(* CODESYS project EL6224_Youtube_Lib.library
   Title: myLibrary
   Version: 0.2
   Placeholder: myLibrary
   Company: soup01

Project tree, tasks and I/O mapping:
  libraries: Tc2_Standard, * (Beckhoff Automation GmbH); Tc2_System, * (Beckhoff Automation GmbH); Tc3_IoLink, * (Beckhoff Automation GmbH); Tc3_Module, * (Beckhoff Automation GmbH); VisuSymbols, 3.5.10.0 (System)
  DUTs/
    data type DUT_ATV320_HMI_NW3_4_PL
    interface ITF_EL6224_Basic: METH_Port_OK
    interface ITF_IDWE_M12MM_NMS_A0: METH_Disable, METH_Update, Prop_ALR, Prop_ALR1, Prop_ALR2, Prop_ALR3, Prop_Enable, Prop_MeasurementValue, Prop_OSS1, Prop_OSS2, Prop_ScalingValue, Prop_StatusWord, Prop_TSS
    interface ITF_LR_TB2000: METH_Update, Prop_Distance, Prop_Enable
  GVLs/
  POUs/
    function block FB_EL6224_Basic [ST]: METH_Port_OK
    function block FB_IDWE_M12MM_NMS_A0 [ST]: METH_Disable, METH_Update, Prop_ALR, Prop_ALR1, Prop_ALR2, Prop_ALR3, Prop_Enable, Prop_MeasurementValue, Prop_OSS1, Prop_OSS2, Prop_ScalingValue, Prop_StatusWord, Prop_TSS
    function block FB_LR_TB2000 [ST]: METH_Update, Prop_Distance, Prop_Enable
  VISUs/
  text list GlobalTextList
*)

// DUTs/DUT_ATV320_HMI_NW3_4_PL
TYPE DUT_ATV320_HMI_NW3_4_PL:
STRUCT
	DIs		:ARRAY[1..6]OF BOOL;
	STO		:BOOL;
END_STRUCT
END_TYPE

// DUTs/ITF_EL6224_Basic
INTERFACE ITF_EL6224_Basic

METHOD METH_Port_OK : BOOL
VAR_INPUT
	iPort		:INT;
END_VAR
END_METHOD

END_INTERFACE

// DUTs/ITF_IDWE_M12MM_NMS_A0
INTERFACE ITF_IDWE_M12MM_NMS_A0

METHOD METH_Disable : BOOL
VAR_INPUT
	iTrigger		:BOOL;
END_VAR
END_METHOD

METHOD METH_Update : BOOL
END_METHOD

PROPERTY Prop_ALR : BOOL
GET
END_GET
END_PROPERTY

PROPERTY Prop_ALR1 : BOOL
GET
END_GET
END_PROPERTY

PROPERTY Prop_ALR2 : BOOL
GET
END_GET
END_PROPERTY

PROPERTY Prop_ALR3 : BOOL
GET
END_GET
END_PROPERTY

PROPERTY Prop_Enable : BOOL
GET
END_GET
END_PROPERTY

PROPERTY Prop_MeasurementValue : INT
GET
END_GET
END_PROPERTY

PROPERTY Prop_OSS1 : BOOL
GET
END_GET
END_PROPERTY

PROPERTY Prop_OSS2 : BOOL
GET
END_GET
END_PROPERTY

PROPERTY Prop_ScalingValue : Byte
GET
END_GET
END_PROPERTY

PROPERTY Prop_StatusWord : byte
GET
END_GET
END_PROPERTY

PROPERTY Prop_TSS : BOOL
GET
END_GET
END_PROPERTY

END_INTERFACE

// DUTs/ITF_LR_TB2000
INTERFACE ITF_LR_TB2000

METHOD METH_Update : BOOL
VAR_INPUT
END_VAR
END_METHOD

PROPERTY Prop_Distance : INT
GET
END_GET
END_PROPERTY

PROPERTY Prop_Enable : BOOL
GET
END_GET
END_PROPERTY

END_INTERFACE

// POUs/FB_EL6224_Basic
FUNCTION_BLOCK FB_EL6224_Basic IMPLEMENTS ITF_EL6224_Basic
VAR_INPUT
END_VAR
VAR_OUTPUT
END_VAR
VAR
	DeviceStatesInputs	AT %I*:ARRAY[1..4]OF USINT;
END_VAR

METHOD METH_Port_OK : BOOL
VAR_INPUT
	iPort	: INT;
END_VAR

METH_Port_OK:=FALSE;

CASE iPort OF
	1..4:
		METH_Port_OK:=DeviceStatesInputs[iPort] = 3;
END_CASE
END_METHOD

END_FUNCTION_BLOCK

// POUs/FB_IDWE_M12MM_NMS_A0
FUNCTION_BLOCK FB_IDWE_M12MM_NMS_A0 IMPLEMENTS ITF_IDWE_M12MM_NMS_A0
VAR_INPUT
	iPortOK		:BOOL;
END_VAR
VAR_OUTPUT
END_VAR
VAR
	//Link to Process Data
		input  AT  %I*:DINT;
		output AT  %Q*:BYTE;
END_VAR

VAR
	StatusWord		:BYTE;
	ScalingValue	:BYTE;
	MesurementValue	:INT;
	InputBuffer		:ARRAY[0..3]OF BYTE;
END_VAR


METHOD METH_Disable : BOOL
VAR_INPUT
	iTrigger	: BOOL;
END_VAR

output.0:=iTrigger;
END_METHOD

METHOD METH_Update : BOOL

StatusWord:=0;
ScalingValue:=0;
MesurementValue:=0;

IF Prop_Enable THEN
	MEMMOVE(
		ADR(InputBuffer)
		,ADR(input)
		,n:=4
	);
		
	MEMMOVE(
		ADR(StatusWord)
		,ADR(InputBuffer)
		,n:=1
	);
	
	MEMMOVE(
		ADR(ScalingValue)
		,ADR(InputBuffer[1])
		,n:=1
		);
	
	MEMMOVE(
		ADR(MesurementValue)
		,ADR(InputBuffer[2])
		,n:=2
		);	
END_IF
END_METHOD

PROPERTY Prop_ALR : BOOL
GET
Prop_ALR:=Prop_ALR1
			OR Prop_ALR2
			OR Prop_ALR3
			;
END_GET
END_PROPERTY

PROPERTY Prop_ALR1 : BOOL
GET
VAR
	_Statusword:BYTE;
END_VAR

_Statusword:=Prop_StatusWord;
Prop_ALR1:=_Statusword.5;
END_GET
END_PROPERTY

PROPERTY Prop_ALR2 : BOOL
GET
VAR
	_Statusword:BYTE;
END_VAR
_Statusword:=Prop_StatusWord;
Prop_ALR2:=_Statusword.6;
END_GET
END_PROPERTY

PROPERTY Prop_ALR3 : BOOL
GET
VAR
	_Statusword:BYTE;
END_VAR
_Statusword:=Prop_StatusWord;
Prop_ALR3:=_Statusword.7;
END_GET
END_PROPERTY

PROPERTY Prop_Enable : BOOL
GET
Prop_Enable:=iPortOK;
END_GET
END_PROPERTY

PROPERTY Prop_MeasurementValue : INT
GET
Prop_MeasurementValue:=MesurementValue;
END_GET
END_PROPERTY

PROPERTY Prop_OSS1 : BOOL
GET
VAR
	_Statusword:BYTE;
END_VAR

_Statusword:=Prop_StatusWord;
Prop_OSS1:=_Statusword.0;
END_GET
END_PROPERTY

PROPERTY Prop_OSS2 : BOOL
GET
VAR
	_Statusword:BYTE;
END_VAR

_Statusword:=Prop_StatusWord;
Prop_OSS2:=_Statusword.1;
END_GET
END_PROPERTY

PROPERTY Prop_ScalingValue : BYTE
GET
Prop_ScalingValue:=ScalingValue;
END_GET
END_PROPERTY

PROPERTY Prop_StatusWord : BYTE
GET
Prop_StatusWord:=StatusWord;
END_GET
END_PROPERTY

PROPERTY Prop_Tss : BOOL
GET
VAR
	_Statusword:BYTE;
END_VAR

_Statusword:=Prop_StatusWord;
Prop_Tss:=_Statusword.2;
END_GET
END_PROPERTY

END_FUNCTION_BLOCK

// POUs/FB_LR_TB2000
FUNCTION_BLOCK FB_LR_TB2000 IMPLEMENTS ITF_LR_TB2000
VAR_INPUT
	iPortOK		:BOOL;
END_VAR
VAR_OUTPUT
END_VAR
VAR
	Inputs	AT %I*:INT;
	Data	:INT;
END_VAR

METHOD METH_Update : BOOL

Data:=0;
IF Prop_Enable THEN
	Data:=Inputs;
END_IF;
END_METHOD

PROPERTY Prop_Distance : INT
GET

Prop_Distance:=0;
IF Prop_Enable THEN
	Prop_Distance:=Data;
END_IF
END_GET
END_PROPERTY

PROPERTY Prop_Enable : BOOL
GET
Prop_Enable:=iPortOK;
END_GET
END_PROPERTY

END_FUNCTION_BLOCK
